// TIA Portal V17 export
// export: Created 2022-06-27T13:58:47.7609257Z, ExportSetting WithDefaults, DisplayName Totally Integrated Automation Portal, DisplayVersion V17 Update 3, DisplayName TIA Portal Openness, DisplayVersion V17 Update 3, DisplayName TIA Portal Version Control Interface, DisplayVersion V17, DisplayName SINAMICS Startdrive Advanced, DisplayVersion V17 Update1, DisplayName SINAMICS Startdrive G110M, G120, G120C, G120D, G120P, G115D, DisplayVersion V17 Update1, DisplayName SINAMICS Startdrive G130, G150, S120, S150, SINAMICS MV, S210, DisplayVersion V17 Update1, DisplayName STEP 7 Professional, DisplayVersion V17 Update 3, DisplayName STEP 7 Safety, DisplayVersion V17, DisplayName WinCC UA Professional, DisplayVersion V17 Update 3
FUNCTION_BLOCK "S062_BUTTONS"   // FB62, LAD
{ S7_Optimized_Access := 'TRUE' }
VERSION : 0.1
// stored: AutoNumber false, IsIECCheckEnabled false, IsRetainMemResEnabled false, MemoryReserve 100, SetENOAutomatically false, UDAEnableTagReadback false
BEGIN

REGION Network 1: S59-2C - Emergency Button Chamber 1
END_REGION

REGION Network 2: S59-3C - Emergency Button Cooler 1
END_REGION

REGION Network 3: S59-4C - Emergency Button Chamber 2
END_REGION

REGION Network 4: S59-5C - Emergency Button Cooler 2
END_REGION

REGION Network 5: S59-6C - Turn off Combustor Button
END_REGION
END_FUNCTION_BLOCK
